# B&R Automation Studio project Bridge_RUC_Motor
Automation Studio 4.9

## Configuration Config1

CPU X90CP172.24-00, AutomationRuntime B4.93, Build 4.1.2, Vc V4.72.6

### Hardware
```
EVE-XCR-C : FBC.0x29C.46342145 v1.153 (OrderNumber=EVE-XCR-C)  [CAN1 -> X90CP172_24_00.IF8 (NodeNumber=32)]
  p200f_connecttomaster = 4
  p2015_connecttomaster = 2
  p2076_connecttomaster = 1
  p2100_parametervalue = 6.7
  p21dc_parametervalue = 0.015
  p21e0_parametervalue = 1.3
  p250a_connecttomaster = 3
  p250a_parametervalue = 2.15
  p250b_connecttomaster = 3
  p250b_parametervalue = 160.8
  p250e_parametervalue = 14
  p250f_parametervalue = -14
  p2511_parametervalue = 0.000454
  p5e49_connecttomaster = 3
  p6061_connecttomaster = 0
  p6064_connecttomaster = 0
  p606c_connecttomaster = 2
  p607a_connecttomaster = 0
  p60ff_connecttomaster = 1
  pheartbeat_producertime = 1000
  p1003_objflags = 1
  p1003sub0_objflags = 1
  p1005_objflags = 1
  p1010_objflags = 1
  p1010sub1_objflags = 1
  p1011_objflags = 1
  p1011sub1_objflags = 1
  p1012_objflags = 1
  p1014_objflags = 1
  p1018_objflags = 1
  p1200_objflags = 1
  p1200sub0_objflags = 1
  p1f50_objflags = 1
  p1f50sub1_objflags = 1
  p1f51_objflags = 1
  p1f51sub1_objflags = 1
  p1f56_objflags = 1
  p1f57_objflags = 1
  p2101_parametervalue = 20
  p2101_objflags = 1
  p2102_parametervalue = 3000
  p2102_objflags = 1
  p2106_parametervalue = 7
  p2106_objflags = 1
  p2109_objflags = 1
  p210a_objflags = 1
  p210b_objflags = 1
  p210c_objflags = 1
  p210d_objflags = 1
  p210e_objflags = 1
  p210f_objflags = 1
  p2110_objflags = 1
  p2111_objflags = 1
  p2112_objflags = 1
  p2113_objflags = 1
  p2114_objflags = 1
  p2120_objflags = 1
  p2121_objflags = 1
  p2122_objflags = 1
  p2123_objflags = 1
  p2124_objflags = 1
  p2125_objflags = 1
  p2126_objflags = 1
  p2127_objflags = 1
  p2128_objflags = 1
  p2129_objflags = 1
  p214f_objflags = 1
  p2150_objflags = 1
  p2151_parametervalue = 1
  p2151_objflags = 1
  p2153_parametervalue = 1
  p2153_objflags = 1
  p2154_objflags = 1
  p2155_parametervalue = 5.36
  p2155_objflags = 1
  p2156_parametervalue = 1000
  p2156_objflags = 1
  p2157_objflags = 1
  p217b_objflags = 1
  p217c_objflags = 1
  p21c8_objflags = 1
  p21e8_parametervalue = 10
  p21e8_objflags = 1
  p21f1_objflags = 1
  p21f2_objflags = 1
  p21f3_objflags = 1
  p21f4_objflags = 1
  p21f5_objflags = 1
  p21f6_objflags = 1
  p21f7_objflags = 1
  p21fb_objflags = 1
  p21fc_objflags = 1
  p21fd_objflags = 1
  p21fe_objflags = 1
  p21ff_objflags = 1
  p2200_objflags = 1
  p2201_objflags = 1
  p2202_objflags = 1
  p2203_objflags = 1
  p22e8_objflags = 1
  p22e9_objflags = 1
  p2360_parametervalue = 1
  p2360_objflags = 1
  p2361_parametervalue = 1
  p2361_objflags = 1
  p2362_parametervalue = 1
  p2362_objflags = 1
  p2364_objflags = 1
  p236f_objflags = 1
  p2370_parametervalue = 29
  p2370_objflags = 1
  p2371_objflags = 1
  p2372_objflags = 1
  p2373_objflags = 1
  p2374_objflags = 1
  p2375_parametervalue = 18
  p2375_objflags = 1
  p2376_parametervalue = 18
  p2376_objflags = 1
  p2377_parametervalue = 11
  p2377_objflags = 1
  p2378_objflags = 1
  p2379_objflags = 1
  p237a_objflags = 1
  p237b_objflags = 1
  p237c_objflags = 1
  p237d_objflags = 1
  p237e_objflags = 1
  p237f_objflags = 1
  p2380_objflags = 1
  p2381_objflags = 1
  p2384_objflags = 1
  p2385_objflags = 1
  p2386_objflags = 1
  p2387_objflags = 1
  p2388_objflags = 1
  p2389_objflags = 1
  p238a_objflags = 1
  p2390_objflags = 1
  p2391_objflags = 1
  p2392_objflags = 1
  p2394_objflags = 1
  p2395_objflags = 1
  p2400_objflags = 1
  p2401_objflags = 1
  p2403_objflags = 1
  p2404_objflags = 1
  p2405_objflags = 1
  p2406_objflags = 1
  p2407_objflags = 1
  p2438_objflags = 1
  p2439_objflags = 1
  p243a_objflags = 1
  p243b_objflags = 1
  p2450_objflags = 1
  p2452_objflags = 1
  p2455_objflags = 1
  p2456_objflags = 1
  p2457_objflags = 1
  p2460_objflags = 1
  p2461_objflags = 1
  p2462_objflags = 1
  p24ff_objflags = 1
  p2500_parametervalue = 1.5
  p2501_parametervalue = 786
  p2502_objflags = 1
  p2503_objflags = 1
  p2504_objflags = 1
  p2505_parametervalue = 1.5
  p2505_objflags = 1
  p2506_parametervalue = 786
  p2507_objflags = 1
  p2508_objflags = 1
  p2509_objflags = 1
  p251b_objflags = 1
  p251c_objflags = 1
  p2521_objflags = 1
  p2522_objflags = 1
  p2530_objflags = 1
  p2531_objflags = 1
  p2532_objflags = 1
  p2533_objflags = 1
  p2538_objflags = 1
  p2539_objflags = 1
  p253a_objflags = 1
  p253b_objflags = 1
  p2540_objflags = 1
  p2541_objflags = 1
  p2542_objflags = 1
  p2543_objflags = 1
  p2548_objflags = 1
  p2549_objflags = 1
  p254a_objflags = 1
  p254b_objflags = 1
  p2550_objflags = 1
  p2551_objflags = 1
  p2552_objflags = 1
  p2553_objflags = 1
  p2558_objflags = 1
  p2559_objflags = 1
  p255a_objflags = 1
  p255b_objflags = 1
  p2560_objflags = 1
  p2561_objflags = 1
  p2562_objflags = 1
  p2563_objflags = 1
  p2568_objflags = 1
  p2569_objflags = 1
  p256a_objflags = 1
  p256b_objflags = 1
  p2570_objflags = 1
  p2571_objflags = 1
  p2572_objflags = 1
  p2573_objflags = 1
  p2578_objflags = 1
  p2579_objflags = 1
  p257a_objflags = 1
  p257b_objflags = 1
  p2580_objflags = 1
  p2581_objflags = 1
  p2582_objflags = 1
  p2583_objflags = 1
  p2588_objflags = 1
  p2589_objflags = 1
  p258a_objflags = 1
  p258b_objflags = 1
  p25fc_objflags = 1
  p25fd_objflags = 1
  p25fe_objflags = 1
  p25ff_objflags = 1
  p2603_objflags = 1
  p2604_objflags = 1
  p2608_objflags = 1
  p2609_objflags = 1
  p260a_objflags = 1
  p260b_objflags = 1
  p260d_objflags = 1
  p260f_objflags = 1
  p2610_objflags = 1
  p2611_objflags = 1
  p2612_objflags = 1
  p2613_objflags = 1
  p2614_objflags = 1
  p2615_objflags = 1
  p2616_objflags = 1
  p2617_objflags = 1
  p2618_objflags = 1
  p2619_objflags = 1
  p261a_objflags = 1
  p261b_objflags = 1
  p261c_objflags = 1
  p261d_objflags = 1
  p2620_objflags = 1
  p2621_objflags = 1
  p2624_objflags = 1
  p262b_objflags = 1
  p262f_objflags = 1
  p2630_objflags = 1
  p2631_objflags = 1
  p2632_objflags = 1
  p2633_objflags = 1
  p2641_objflags = 1
  p2642_objflags = 1
  p2643_objflags = 1
  p2644_objflags = 1
  p2645_objflags = 1
  p2646_objflags = 1
  p264e_objflags = 1
  p26db_objflags = 1
  p26dc_objflags = 1
  p26dd_objflags = 1
  p26df_objflags = 1
  p26e4_objflags = 1
  p26e5_objflags = 1
  p2743_objflags = 1
  p5820_objflags = 1
  p5820sub1_objflags = 1
  p5820sub2_objflags = 1
  p5820sub3_objflags = 1
  p58aa_objflags = 1
  p5e4b_objflags = 1
  p5e4e_objflags = 1
  p5e80_objflags = 1
  p5ec5_objflags = 1
  p5edb_objflags = 1
  p5edc_objflags = 1
  p5ede_objflags = 1
  p5ee4_objflags = 1
  p6007_objflags = 1
  p605a_objflags = 1
  p605d_objflags = 1
  p607b_objflags = 1
  p607d_objflags = 1
  p6098_objflags = 1
  p6099_objflags = 1
  p60c2_objflags = 1
X90CP172_24_00 : X90CP172.24-00 v1.4.6.0  [X1 -> X1a.SL]
  Module X1a (Type=X1, Virtual=true, Version=1.4.6.0)
    Connection (Connector=SL, TargetModule=X90CP172_24_00, TargetConnector=X1)
  Connector IF2:
    ActivateDevice = 1
  Connector IF8:
    Baudrate = 250000
    ActivateCANIO = 0
    ActivateCanOpen = 1
  ConfigurationID = Bridge_RUC_Motor_Config1
  Cyclic1Duration = 10000
  Cyclic1Tolerance = 10000
  Cyclic2Duration = 20000
  Cyclic2Tolerance = 20000
  Cyclic3Duration = 50000
  Cyclic3Tolerance = 50000
  Cyclic4Duration = 100000
  Cyclic4Tolerance = 100000
  Cyclic5Duration = 200000
  Cyclic5Tolerance = 200000
  Cyclic6Duration = 500000
  Cyclic6Tolerance = 500000
  Cyclic7Duration = 1000000
  Cyclic7Tolerance = 1000000
  Cyclic8Duration = 10000
  Cyclic8Tolerance = 30000000
  FileDevice1
  FileDeviceName1 = USER
  FileDevicePath1 = USER_PATH
```

### IoMap.iom - X90CP172_24_00/IoMap.iom
```iecst
VAR_CONFIG
	::ServoCtrl:ServoDriveModuleOK AT %IX."EVE-XCR-C".ModuleOk;
	::ServoCtrl:IOOperationModeDisplay AT %IW."EVE-XCR-C".OperationModeDisplay_2015;
	::ServoCtrl:IOControlWord AT %QW."EVE-XCR-C".ControlWord_6040;
	::ServoCtrl:IOStatusWord AT %IW."EVE-XCR-C".StatusWord_6041;
	::ServoCtrl:IOOperationMode AT %QB."EVE-XCR-C".OperationMode_6060;
	::ServoCtrl:IOVelocitySetpoint AT %QD."EVE-XCR-C".VelocitySet_point_60FF;
	::ServoCtrl:IOActualVelocity AT %ID."EVE-XCR-C".ActualVelocity_606C;
	::ServoCtrl:VelocityLoopKp AT %QD."EVE-XCR-C".VelocityLoopKp_250A;
	::ServoCtrl:VelocityLoopKi AT %QD."EVE-XCR-C".VelocityLoopKi_250B;
END_VAR
```

## Logical view

Binary libraries used (declarations not repeated): AsCANopen, AsBrStr, operator, runtime, astime, AsIecCon, ArCan, standard

### Global.typ - Global data types
```iecst
TYPE
	ServoData_typ : 	STRUCT
		VelocitySetPoint : DINT; (*[rpm]*)
		VelocityActual : DINT; (*[rpm]*)
		ServoON : BOOL;
		Servo_OK : BOOL;
	END_STRUCT;
END_TYPE
```

### Global.var - Global variables
```iecst
VAR
	gServoData : ServoData_typ;
END_VAR
```


### Program Logical/ServoCtrl (ANSIC)

#### Types.typ
```iecst
TYPE
	SDO_step_type :
		(
		SDO_SET_REGISTERS,
		SDO_WAIT_4_CMD,
		SDO_RUN_TIMER,
		SDO_READ,
		SDO_WRITE_MAX_CURRENT,
		SDO_WRITE_MAX_VELOCITY,
		SDO_WRITE_MAX_ACCELERATION,
		SDO_WRITE_MAX_DECELERATION,
		SDO_WRITE_VELOCITY_FEEDBACK,
		SDO_WRITE_2500,
		SDO_WRITE_2501,
		SDO_WRITE_2505,
		SDO_WRITE_2506,
		SDO_WRITE_250A,
		SDO_WRITE_250B
		);
	SDO_type : 	STRUCT
		step : SDO_step_type;
		device : STRING[80];
		CANopenSDORead8_0 : CANopenSDORead8;
		CANopenSDOWrite8_0 : CANopenSDOWrite8;
	END_STRUCT;
	test_type : 	STRUCT
		data0 : USINT;
		data1 : USINT;
		data2 : USINT;
		data3 : USINT;
	END_STRUCT;
	SERVO_type : 	STRUCT
		step : SERVO_step_type;
		EnableOperation : BOOL;
		DisableOperation : BOOL;
		ActualVelocity : DINT; (*[mrev/s]*)
	END_STRUCT;
	SERVO_step_type :
		(
		SERVO_INIT,
		SERVO_FIRST_STEP,
		SERVO_SWITCH_ON_DISABLED,
		SERVO_READY_TO_SWITCH_ON,
		SERVO_SWITCHED_ON,
		SERVO_OPERATION_ENABLE
		);
END_TYPE
```

#### Variables.var
```iecst
VAR
	ArCanSetBitTimingRegisters_0 : ArCanSetBitTimingRegisters;
	SDO : SDO_type := (0);
	Test : REAL;
	MaxCurrent : REAL := 14.6; (*[A]*)
	VelocityLoopKi : REAL := 14;
	VelocityLoopKp : REAL := 1.5;
	ProfilerMaxVelocity : REAL := 3; (*[rev/s]*)
	ProfilerMaxAcc : REAL := 5; (*[rev/s2]*)
	ProfilerMaxDec : REAL := 5; (*[rev/s2]*)
	VelocityFeedbackFilter : UDINT := 100;
	TON_0 : TON;
	ParamWriteDone : BOOL;
	SDOWriteWaitTime : TIME := 10000; (*[ms]*)
	ServoDriveModuleOK : BOOL;
	IOControlWord : UINT;
	IOStatusWord : UINT;
	IOOperationMode : SINT;
	IOVelocitySetpoint : DINT; (*[mrev/s]*)
	IOOperationModeDisplay : UINT;
	IOActualVelocity : DINT; (*[mrev/s]*)
	SERVO : SERVO_type;
	mask0 : USINT := 1;
	mask1 : USINT := 2;
	mask2 : USINT := 4;
	mask3 : USINT := 8;
	mask4 : USINT := 16;
	mask5 : USINT := 32;
	mask6 : USINT := 64;
	mask7 : USINT := 128;
END_VAR
```

#### Main.c
```c
#include <bur/plctypes.h>

#ifdef _DEFAULT_INCLUDES
	#include <AsDefault.h>
#endif

#define TRUE 1
#define FALSE 0
#define MAX(x, y) (((x) > (y)) ? (x) : (y))
#define MIN(x, y) (((x) < (y)) ? (x) : (y))
#define abs(x) ((x)<0 ? -(x) : (x))

void _INIT ProgramInit(void)
{
	SDO.step = SDO_SET_REGISTERS;
	brsstrcpy((UDINT) SDO.device, (UDINT) "IF8");  //set interface
	gServoData.Servo_OK = FALSE;
}

BOOL Ready_to_switch_on_disabled_state (void){ // 592
	return ((IOStatusWord & mask6) && (~IOStatusWord & mask3) && (~IOStatusWord & mask2) && (~IOStatusWord & mask1) && (~IOStatusWord & mask0));
}

void _CYCLIC ProgramCyclic(void)
{

		// ============== STATE MACHINE FOR WRITING SERVO PARAMETERS ("SDO download") ==============
		switch(SDO.step) {

			case SDO_SET_REGISTERS :

				ArCanSetBitTimingRegisters_0.Execute = 1;
				brsstrcpy((UDINT) &ArCanSetBitTimingRegisters_0.DeviceName, (UDINT) &SDO.device);
				ArCanSetBitTimingRegisters_0.Register0 = 0x01; 	/*250kbit/s*/	/* 0x00; Set to 1 000 000 bit/s */
				ArCanSetBitTimingRegisters_0.Register1 = 0x1C; 	/*250kbit/s*/	/* 0x14; Set to 1 000 000 bit/s */

				ArCanSetBitTimingRegisters(&ArCanSetBitTimingRegisters_0);

				if (ArCanSetBitTimingRegisters_0.Done) SDO.step = SDO_WAIT_4_CMD;

				break;
			case SDO_WAIT_4_CMD:

				if (ServoDriveModuleOK && !ParamWriteDone) {
					SDO.step = SDO_RUN_TIMER;
				}
				break;

			case SDO_RUN_TIMER:

				TON_0.PT = SDOWriteWaitTime;
				TON_0.IN = 1;

				if (TON_0.Q) {
					TON_0.IN = 0;
					SDO.step = SDO_READ;
				}
				break;

			case SDO_READ:

				SDO.CANopenSDORead8_0.enable = 1;
				SDO.CANopenSDORead8_0.pDevice =(UDINT) &(SDO.device);
				SDO.CANopenSDORead8_0.node = 32; //(* Node ID from IO device *)
				SDO.CANopenSDORead8_0.index = 0x21E0;
				SDO.CANopenSDORead8_0.subindex = 0x00;

				CANopenSDORead8(&SDO.CANopenSDORead8_0); // (* Call function block *)

				if (SDO.CANopenSDORead8_0.status == ERR_OK) {
					brsmemcpy((UDINT) &Test, (UDINT) &SDO.CANopenSDORead8_0.data0, 4);
					SDO.step = SDO_WRITE_MAX_CURRENT; //(* next step *)
				} else if (SDO.CANopenSDORead8_0.status == ERR_FUB_BUSY) { // (* FBK not yet finished *)
					//busy
				} else {  //(* Error step *)
					//	SDO.step = 10;
				}
				break;

			case SDO_WRITE_MAX_CURRENT:

				SDO.CANopenSDOWrite8_0.enable = 1;
				SDO.CANopenSDOWrite8_0.pDevice = (UDINT) &(SDO.device);
				SDO.CANopenSDOWrite8_0.node = 32;  //(* Node ID from IO device *)
				SDO.CANopenSDOWrite8_0.index = 0x21E0;
				SDO.CANopenSDOWrite8_0.subindex = 0x00;
				brsmemcpy((UDINT) &SDO.CANopenSDOWrite8_0.data0, (UDINT) &MaxCurrent, 4);
				SDO.CANopenSDOWrite8_0.datalen = 4;

				if (SDO.CANopenSDOWrite8_0.status == ERR_OK) { // (* OK *)
					SDO.step = SDO_WRITE_MAX_VELOCITY; //(* next step *)
				} else if (SDO.CANopenSDOWrite8_0.status == ERR_FUB_BUSY) { // (* FBK not yet finished *)
					//(* busy *)
				} else { // (* Error step *)
					//	SDO.step = 10;
				}
				break;

			case SDO_WRITE_MAX_VELOCITY:

				SDO.CANopenSDOWrite8_0.enable = 1;
				SDO.CANopenSDOWrite8_0.pDevice = (UDINT) &(SDO.device);
				SDO.CANopenSDOWrite8_0.node = 32;  //(* Node ID from IO device *)
				SDO.CANopenSDOWrite8_0.index = 0x2025;
				SDO.CANopenSDOWrite8_0.subindex = 0x00;
				brsmemcpy((UDINT) &SDO.CANopenSDOWrite8_0.data0, (UDINT) &ProfilerMaxVelocity, 4);
				SDO.CANopenSDOWrite8_0.datalen = 4;

				if (SDO.CANopenSDOWrite8_0.status == ERR_OK) { // (* OK *)
					SDO.step = SDO_WRITE_MAX_ACCELERATION; //(* next step *)
				} else if (SDO.CANopenSDOWrite8_0.status == ERR_FUB_BUSY) { // (* FBK not yet finished *)
					//(* busy *)
				} else { // (* Error step *)
					//	SDO.step = 10;
				}
				break;

			case SDO_WRITE_MAX_ACCELERATION:

				SDO.CANopenSDOWrite8_0.enable = 1;
				SDO.CANopenSDOWrite8_0.pDevice = (UDINT) &(SDO.device);
				SDO.CANopenSDOWrite8_0.node = 32;  //(* Node ID from IO device *)
				SDO.CANopenSDOWrite8_0.index = 0x2026;
				SDO.CANopenSDOWrite8_0.subindex = 0x00;
				brsmemcpy((UDINT) &SDO.CANopenSDOWrite8_0.data0, (UDINT) &ProfilerMaxAcc, 4);
				SDO.CANopenSDOWrite8_0.datalen = 4;

				if (SDO.CANopenSDOWrite8_0.status == ERR_OK) { // (* OK *)
					SDO.step = SDO_WRITE_MAX_DECELERATION; //(* next step *)
				} else if (SDO.CANopenSDOWrite8_0.status == ERR_FUB_BUSY) { // (* FBK not yet finished *)
					//(* busy *)
				} else { // (* Error step *)
					//	SDO.step = 10;
				}
				break;

			case SDO_WRITE_MAX_DECELERATION:

				SDO.CANopenSDOWrite8_0.enable = 1;
				SDO.CANopenSDOWrite8_0.pDevice = (UDINT) &(SDO.device);
				SDO.CANopenSDOWrite8_0.node = 32;  //(* Node ID from IO device *)
				SDO.CANopenSDOWrite8_0.index = 0x2027;
				SDO.CANopenSDOWrite8_0.subindex = 0x00;
				brsmemcpy((UDINT) &SDO.CANopenSDOWrite8_0.data0, (UDINT) &ProfilerMaxDec, 4);
				SDO.CANopenSDOWrite8_0.datalen = 4;

				if (SDO.CANopenSDOWrite8_0.status == ERR_OK) { // (* OK *)
					SDO.step = SDO_WRITE_VELOCITY_FEEDBACK; //(* next step *)
				} else if (SDO.CANopenSDOWrite8_0.status == ERR_FUB_BUSY) { // (* FBK not yet finished *)
					//(* busy *)
				} else { // (* Error step *)
					//	SDO.step = 10;
				}
				break;

			case SDO_WRITE_VELOCITY_FEEDBACK:

				SDO.CANopenSDOWrite8_0.enable = 1;
				SDO.CANopenSDOWrite8_0.pDevice = (UDINT) &(SDO.device);
				SDO.CANopenSDOWrite8_0.node = 32;  //(* Node ID from IO device *)
				SDO.CANopenSDOWrite8_0.index = 0x2551;
				SDO.CANopenSDOWrite8_0.subindex = 0x00;
				brsmemcpy((UDINT) &SDO.CANopenSDOWrite8_0.data0, (UDINT) &VelocityFeedbackFilter, 4);
				SDO.CANopenSDOWrite8_0.datalen = 4;

				if (SDO.CANopenSDOWrite8_0.status == ERR_OK) { // (* OK *)
					ParamWriteDone = 1;
					SDO.step = SDO_WAIT_4_CMD; //(* next step *)
				} else if (SDO.CANopenSDOWrite8_0.status == ERR_FUB_BUSY) { // (* FBK not yet finished *)
					//(* busy *)
				} else { // (* Error step *)
					//	SDO.step = 10;
				}
				break;
		}

		// If servo drive module is not OK, get ready to write servo parameters again
		if (!ServoDriveModuleOK) {
			ParamWriteDone = 0;
			SDO.step = SDO_WAIT_4_CMD;
			gServoData.Servo_OK = FALSE;
		}
		else
			gServoData.Servo_OK = TRUE;

		CANopenSDOWrite8(&SDO.CANopenSDOWrite8_0); //call function block
		SDO.CANopenSDOWrite8_0.enable = 0; //disable function block

		TON(&TON_0); //call function block
		TON_0.IN = 0; //disable function block

		// Copy data
		//	gServoData.VelocityActual =(DINT) (((REAL) IOActualVelocity / 1000.0) * 60.0);
		gServoData.VelocityActual = (DINT) ((REAL) IOActualVelocity /** SERVO_VELOCITY_RECALC_PARAM*/);

		// Enable/disable servo drive
		if ((SERVO.step == SERVO_SWITCHED_ON) && (gServoData.ServoON)) {
			SERVO.EnableOperation = 1;
		}
		if ((SERVO.step == SERVO_OPERATION_ENABLE) && (!gServoData.ServoON)) {
			SERVO.DisableOperation = 1;
		}

		// ============== STATE MACHINE FOR SERVO DRIVE CONTROL ==============================
		switch(SERVO.step) {

			case SERVO_INIT:

				IOControlWord = 0; //Disable voltage command

				if (ParamWriteDone) {
					SERVO.step = SERVO_FIRST_STEP;
				}
				break;

			case SERVO_FIRST_STEP:

				IOControlWord = 0; //Disable voltage command

				if (Ready_to_switch_on_disabled_state()) { //0bxxxx xxxx x1xx 0000 (592 decimalne)
					SERVO.step = SERVO_SWITCH_ON_DISABLED;
				}
				break;

			case SERVO_SWITCH_ON_DISABLED:

				IOControlWord = 6; //Shutdown command

				if ((~IOStatusWord & mask6) && (IOStatusWord & mask5) && (~IOStatusWord & mask3) && (~IOStatusWord & mask2) && (~IOStatusWord & mask1) && (IOStatusWord & mask0)) { //0bxxxx xxxx x01x 0001
					SERVO.step = SERVO_READY_TO_SWITCH_ON;
				}
				break;

			case SERVO_READY_TO_SWITCH_ON:

				IOControlWord = 7; //Switch on command

				if ((~IOStatusWord & mask6) && (IOStatusWord & mask5) && (~IOStatusWord & mask3) && (~IOStatusWord & mask2) && (IOStatusWord & mask1) && (IOStatusWord & mask0)) { //0bxxxx xxxx x01x 0011
					SERVO.step = SERVO_SWITCHED_ON;
				}
				break;

			case SERVO_SWITCHED_ON:

				IOOperationMode = 3; //Velocity mode

				if (SERVO.EnableOperation) {
					IOControlWord = 15; //Enable operation command
				}

				if ((~IOStatusWord & mask6) && (IOStatusWord & mask5) && (~IOStatusWord & mask3) && (IOStatusWord & mask2) && (IOStatusWord & mask1) && (IOStatusWord & mask0)) { //0bxxxx xxxx x01x 0111
					IOVelocitySetpoint = 0;
					SERVO.step = SERVO_OPERATION_ENABLE;
				}

				if (Ready_to_switch_on_disabled_state()) { //0bxxxx xxxx x1xx 0000 // 592
					SERVO.step = SERVO_SWITCH_ON_DISABLED;
				}

				break;

			case SERVO_OPERATION_ENABLE:

				IOVelocitySetpoint = (DINT) ((REAL) gServoData.VelocitySetPoint /*/ SERVO_VELOCITY_RECALC_PARAM*/);

				if (SERVO.DisableOperation) {
					IOControlWord = 7; //Switch on command
					SERVO.step = SERVO_SWITCHED_ON;
				}

				if (Ready_to_switch_on_disabled_state()) { //0bxxxx xxxx x1xx 0000 // 592
					SERVO.step = SERVO_SWITCH_ON_DISABLED;
				}

				break;
		}

		// Reset commands
		SERVO.EnableOperation = 0;
		SERVO.DisableOperation = 0;

}

void _EXIT ProgramExit(void)
{

}
```

### GLOBAL_DEFINES.h
```c
#ifndef __GLOBAL_DEFINES__
#define __GLOBAL_DEFINES__

//#define _DEBUG								//WARNING: DEBUG causes a malfunction -\_(-.-)_/-
//#define _FALLBACK_FORCE

#ifdef _DEBUG
	#define SWVERSION "       "
#else
	#define SWVERSION "       "
#endif

#define TRUE 1
#define FALSE 0
#define MAX(x, y) (((x) > (y)) ? (x) : (y))
#define MIN(x, y) (((x) < (y)) ? (x) : (y))
#define abs(x) ((x)<0 ? -(x) : (x))
#define PWM_MAX 32767
#define PP_RATIO 0.007246

#endif
```
